Fanuc KAREL source: kt00525.KL

-- PROVISIONAL review KL for V770-1; original PC SHA256 e76d01c245b02d131ee915dd8b6877f8a960eb2d12cebb85d480aa84186db697
-- Incomplete behavior may be omitted. Consult companion uncertainty JSON. Do not deploy.
PROGRAM KT00525
%NOLOCKGROUP
-- UNRESOLVED_DECL P1 type=000106
-- UNRESOLVED_DECL P2 type=000106
-- UNRESOLVED_DECL OUT type=000102
BEGIN
  -- UNRESOLVED_PC offsets 5-20; opcodes 2E,22,32,35
  -- UNRESOLVED_PC offsets 25-40; opcodes 2E,22,32,35
  -- UNRESOLVED_PC offsets 45-60; opcodes 2E,22,32,35
  -- UNRESOLVED_PC offsets 65-80; opcodes 2E,22,32,35
  -- UNRESOLVED_PC offsets 85-124; opcodes 49,7E,49,7E,60,7E,4A
  -- UNRESOLVED_PC offsets 129-133; opcodes 7F
END KT00525
